Staubli VAL3: OUT.pjx

--- OUT.pjx ---
Parameters version=s7.5 stackSize=5000 millimeterUnit=true
Program file=find.pgx
Program file=get.pgx
Program file=getAnaValue.pgx
Program file=getItem.pgx
Program file=getSize.pgx
Program file=getStatus.pgx
Program file=insert.pgx
Program file=isActive.pgx
Program file=isEnable.pgx
Program file=load.pgx
Program file=onEdit.pgx
Program file=onInsert.pgx
Program file=onProgEnd.pgx
Program file=onRun.pgx
Program file=onStart.pgx
Program file=onStop.pgx
Program file=reset.pgx
Program file=save.pgx
Program file=setActive.pgx
Program file=setAnaValue.pgx
Program file=setEnable.pgx
Program file=setItem.pgx
Program file=setStatus.pgx
Data file=OUT.dtx
Library alias=saveInOut path=Disk://saveInputOutput/saveInputOutput.pjx
Library alias=saveData path=Disk://saveData/saveData.pjx
Library alias=use path=Disk://kernel/userPage/userPage.pjx
Library alias=cycleStatus path=Disk://cycleStatus/cycleStatus.pjx
Library alias=language path=Disk://kernel/language/language.pjx
Type name=dioItem path=Disk://kernel/template/dioItem/dioItem.pjx
Type name=aioItem path=Disk://kernel/template/aioItem/aioItem.pjx

--- OUT.dtx ---
public string sItems
string sMessage
string sKey

--- find.pgx ---
public program find(string& x_sItem[], bool& x_bFound[])
  local num i
  local num l_nSize
  local string l_sItem
begin
  // find an item in the list
  x_bFound=isDefined(saveInOut:dOutput[x_sItem])

end

--- get.pgx ---
public program get(string& x_sItem[], num x_nIndex)
  local num l_nSize
  local string l_sKey
  local num i
begin
  x_sItem=sKey[x_nIndex]
end

--- getAnaValue.pgx ---
public program getAnaValue(num& x_nValue[], num x_nIndex)
begin
  x_nValue=aioGet(saveInOut:aio_out[x_nIndex])
end

--- getItem.pgx ---
public program getItem(string& x_sItem, string& x_sId)
begin
  // get the name
  x_sItem=saveInOut:dOutput[x_sId].sName
end

--- getSize.pgx ---
public program getSize(num& x_nSize[])
begin
  // size
  x_nSize=size(saveInOut:dOutput)
end

--- getStatus.pgx ---
public program getStatus(bool& x_bStatus[], string x_sItem)
  local num l_nSize
begin
  // give back the status
  x_bStatus=saveInOut:dOutput[x_sItem].dDio
end

--- insert.pgx ---
public program insert(string x_sItem, bool& x_bDone)
begin
  // insert a new item
  if isDefined(saveInOut:dOutput[x_sItem])==false
    x_bDone=true
    insert(saveInOut:dOutput[x_sItem])
  else
    // already exist
    x_bDone=false
  endIf

end

--- isActive.pgx ---
public program isActive(bool& x_bActive[], string x_sItem)
  local num l_nSize
begin
  // check if is active
  x_bActive=saveInOut:dOutput[x_sItem].bActive
end

--- isEnable.pgx ---
public program isEnable(bool& x_bEnable[], string x_sItem)
  local num l_nSize
begin
  // check if is active
  x_bEnable=saveInOut:dOutput[x_sItem].bEnable
end

--- onEdit.pgx ---
public program onEdit(string& x_sItem[])
  local string l_sItem[3]
  local num l_nCount
  local string l_sFlag[3]
  local string l_sName[3]
  local num i
  local string l_sData
  local num l_nFlag
  local string l_sMessage
  local string l_sId
begin
  // show the real name
  l_sData=x_sItem
  do
    // sMode
    i=find(l_sData,"AND")
    if i!=-1
      i=i+len("AND")+1
    endIf
    //
    if i!=-1
      l_sItem[l_nCount]=left(l_sData,i)
      l_sData=right(l_sData,len(l_sData)-i)
    else
      l_sItem[l_nCount]=l_sData
    endIf
    l_nFlag=find(l_sItem[l_nCount],">")
    // l_bMode
    if find(l_sItem[l_nCount],">ON")!=-1
      l_sFlag[l_nCount]=">ON"+chr(10)
    else
      l_sFlag[l_nCount]=">OFF"+chr(10)
    endIf
    // sItem
    l_sItem[l_nCount]=left(l_sItem[l_nCount],l_nFlag)
    l_sId=l_sItem[l_nCount]
    l_sName[l_nCount]=saveInOut:dOutput[l_sId].sName
    l_nCount=l_nCount+1
  until i==-1
  // show the ID+name
  l_sMessage=""
  for i=0 to 2
    if l_sItem[i]!=""
      l_sMessage=l_sMessage+l_sItem[i]+"["+l_sName[i]+"]"+l_sFlag[i]
    endIf
  endFor
  // popUp IT
  popUpMsg(l_sMessage)
end

--- onInsert.pgx ---
public program onInsert(string& x_sItem[])
  local num l_nSize
  local string l_sEvent
  local num i
  local num l_nKey
  local string l_sMessage
  local bool l_bActive
  local num l_nIndex
  local string l_sItemList
  local num l_nSizeList
  local string l_sButton
  local string l_sKey
  local string l_sName
  local string l_sItem
begin
  x_sItem=""
  call getSize(l_nSizeList)
  do
    // create the list
    //
    call use:setSizeList(10,0,28,11)
    call use:listcreate("OUTPUT ")
    // start from the first
    l_sKey=first(saveInOut:dOutput)
    while l_sKey!=""
      // scan
      call isActive(l_bActive,l_sKey)
      if l_bActive
        // insert into the list
        l_sName=saveInOut:dOutput[l_sKey].sName
        l_sItemList=l_sKey+" {"+l_sName+"}"
        call use:listadd(l_sItemList)
      endIf
      // next
      l_sKey=next(saveInOut:dOutput[l_sKey])
    endWhile
    //
    // display the list
    //
    call use:listredraw(min(l_nIndex-use:nView,0))
    //
    // wait a KEY
    //
    do
      l_nKey=get()
      // get one input from the list
      call use:listevent(l_nKey,l_nIndex,l_sEvent)
      if l_nKey==255
        return
      endIf
    until l_nKey==270
    //
    // insert the sentence
    //
    if l_sEvent==""
      return
    else
      l_sEvent=left(l_sEvent,find(l_sEvent,"{")-1)
    endIf
    // update
    l_sItem=l_sItem+l_sEvent
    // get the status ON-OFF
    call use:stringToArray("ON,OFF",sMessage)
    call language:message(l_sMessage,40)
    call use:questionDialog(l_sMessage,sMessage,i)
    if i==1
      l_sItem=l_sItem+">ON"
    else
      if i==2
        l_sItem=l_sItem+">OFF"
      else
        // escape
        return
      endIf
    endIf
    l_nSize=l_nSize+1
    // define the operator
    if l_nSize!=3
      call language:message(l_sMessage,41)
      l_sButton="AND"
      call use:questionDialog(l_sMessage,l_sButton,i)
      if i==-1
        // escape
        return
      else
        if i==1
          l_sItem=l_sItem+" AND "
        endIf
      endIf
    endIf
  until i==0 or l_nSize==3
  // give it back
  x_sItem=l_sItem
end

--- onRun.pgx ---
public program onRun(string& x_sItem[])
  local num l_nCount
  local string l_sItem[3]
  local num l_nFlag
  local bool l_bMode[3]
  local bool l_bActive
  local bool l_bFound
  local num l_nSize
  local num i
  local num j
  local string l_sName
  local string l_sMessage
begin
  //
  // find how many time and fill sItem and l_bMode
  //
  l_nCount=-1
  do
    l_nCount=l_nCount+1
    // sMode
    i=find(x_sItem,"AND")
    if i!=-1
      i=i+len("AND")+1
    endIf
    //
    if i!=-1
      l_sItem[l_nCount]=left(x_sItem,i)
      x_sItem=right(x_sItem,len(x_sItem)-i)
    else
      l_sItem[l_nCount]=x_sItem
    endIf
    l_nFlag=find(l_sItem[l_nCount],">")
    // l_bMode
    if find(l_sItem[l_nCount],">ON")!=-1
      l_bMode[l_nCount]=true
    else
      l_bMode[l_nCount]=false
    endIf
    //sItem
    l_sItem[l_nCount]=left(l_sItem[l_nCount],l_nFlag)
  until i==-1
  //
  // set the OUTPUT wait for the output
  //
  call getSize(l_nSize)
  for i=0 to l_nCount
    // execute
    l_sName=l_sItem[i]
    if saveInOut:dOutput[l_sName].bEnable
      saveInOut:dOutput[l_sName].dDio=l_bMode[i]
    endIf
  endFor
end

--- onStart.pgx ---
public program onStart(string& x_sItem[])
// check and put all the boolean as the status of BIO-MIO-MODBUS-FIELDBUS-ARMIO
  local num i
  local num l_nModbusOut
  local num l_nFieldbusOut
  local bool l_bChange
  local num l_nResult
  local string l_sPath
  local bool l_bCheck
  local string l_sKey
begin
  if x_sItem=="init"
    //
    // DIGITAL INPUT
    //
    // set the default value
    call saveInOut:setOutput(0)
//    // BIO
//    call saveInOut:setOutput(1)
//    // BIO2 - MIO
//    call saveInOut:setOutput(2)
//    // MODBUS
//    call saveInOut:setOutput(3)
//    // USER
//    call saveInOut:setOutput(4)
//    // REMIO
    //    call saveInOut:setOutput(5)
    call saveInOut:setOutput(6)
    //
    // SAVE
    //
    call save(l_nResult)
    if l_nResult==0
      logMsg("[KERNEL] SUPERVISOR>Output: Save Done")
    else
      logMsg("error "+toString("",l_nResult)+" saving the saveInputOutput")
      popUpMsg("error "+toString("",l_nResult)+" saving the saveInputOutput")
    endIf
  endIf
  // build the list for easy access
  // start from the first
  resize(sKey,1,1)
  sKey=""
  if isDefined(saveInOut:dOutput["valve1"])
    sKey[0]="valve1"
  endIf
  if isDefined(saveInOut:dOutput["valve2"])
    append(sKey)
    sKey[1]="valve2"
  endIf
  if isDefined(saveInOut:dOutput["fOut0"])
    append(sKey)
    sKey[2]="fOut0"
  endIf
  l_sKey=first(saveInOut:dOutput)
  i=size(sKey)-1
  // search it
  //
  while l_sKey!=""
    if find(l_sKey,"valve")==-1 and find(l_sKey,"fOut")==-1
      if !(sKey[0]=="" and i==0)
        append(sKey)
        i=i+1
      endIf
      sKey[i]=l_sKey
    endIf
    l_sKey=next(saveInOut:dOutput[l_sKey])
  endWhile
end

--- onStop.pgx ---
public program onStop(string& x_sItem[])
begin
end

--- save.pgx ---
public program save(num& x_nResult[])
begin
  x_nResult=saveInOut:libSave()
  if x_nResult!=0
    delay(0.5)
    x_nResult=saveInOut:libSave()
  endIf
end

--- setActive.pgx ---
public program setActive(bool x_bActive, string x_sItem)
  local num l_nSize
begin
  // check if is active
  saveInOut:dOutput[x_sItem].bActive=x_bActive
end

--- setAnaValue.pgx ---
public program setAnaValue(num x_nValue, string x_sItem)
begin
  // set the value in to the AIO
  aioSet(saveInOut:aOutput[x_sItem].aAio,x_nValue)
end

--- setEnable.pgx ---
public program setEnable(bool x_bEnable, string x_sItem)
  local num l_nSize
begin
  // check if is active
  saveInOut:dOutput[x_sItem].bEnable=x_bEnable
end

--- setItem.pgx ---
public program setItem(string x_sItem, string& x_sId[])
  local num l_nSize
begin
  // set the ITEM name
  saveInOut:dOutput[x_sId].sName=x_sItem
end

--- setStatus.pgx ---
public program setStatus(bool x_bStatus, string x_sId)
begin
  // change the BIT status
  saveInOut:dOutput[x_sId].dDio=x_bStatus
end
